Staubli VAL3: pickSample.pgx

program pickSample()
begin
  taskCreate "notGrip",100,notGrip()
  currentSamPosJ=herej()
  currentSamPos=jointToPoint(flange,world,currentSamPosJ)
  movel(appro(currentSamPos,{0,0,80,0,0,0}),flange,mNomSpeed)
  waitEndMove()
  taskKill("notGrip")
  switchGripper=true
  movel(appro(currentSamPos,{0,0,0,0,0,0}),flange,mNomSpeed)
  waitEndMove()
  message="pickSample:done"
  taskCreate "sendStatus",100,sendStatus()
  taskKill("pickSample")
  //taskKill("notGrip")
end
